TYPE STMInfoData :
STRUCT
	infoData1 : UINT;
	infoData2 : UINT;
	infoData3 : UINT;
END_STRUCT
END_TYPE

(* stored: Version 1.1.0.1, ProductVersion 3.1.4024.11
   DUT STMInfoData: Id {efade9f3-8636-4785-b0f9-ed49feab9d7e} *)
